// TIA Portal V19 export
FUNCTION_BLOCK "Arduino_Modbus"   // FB6, LAD
{ S7_Optimized_Access := 'TRUE' }
// v0.0.1 has not been tested
// stored: MemoryReserve 100, SetENOAutomatically false
   VAR_INPUT
      Proces_Item : Bool;
      Place_Item_Conveyor : Bool;
      Place_Item_Storage : Bool;
      Scrap_Item : Bool;
      Speed_Transport : Int := 10;
      Speed_Grinding : Int := 10;
      Grinding_Coordinates : Bool;
      Letter : DB_ANY;
   END_VAR
   VAR_OUTPUT
      Working : Bool;
      Done : Bool;
      Error : Bool;
      Reached_Coordinates : Bool;
   END_VAR
   VAR
      DISCONNECT : Bool;
      Address : TCON_IP_v4;
      ReceiveData : Array[0..5] of Int;
      SendData : Array[0..5] of Int;
   END_VAR
   // Address.InterfaceId := 64;
   // Address.ID := 1;
   // Address.ConnectionType := 11;
   // Address.ActiveEstablished := TRUE;
   // Address.RemoteAddress.ADDR[1] := 192;
   // Address.RemoteAddress.ADDR[2] := 168;
   // Address.RemoteAddress.ADDR[3] := 1;
   // Address.RemoteAddress.ADDR[4] := 61;
   // Address.RemotePort := 502;
   // Address.LocalPort := 502;
BEGIN

REGION Network 1: MB_CLIENT
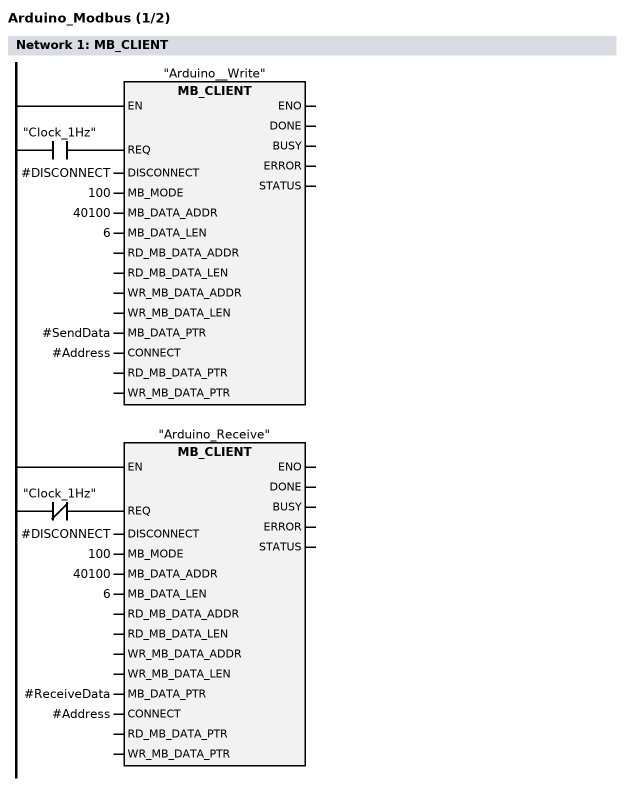
   RUNG wire#powerrail
      "Arduino__Write".MB_CLIENT(REQ := wire#w1, DISCONNECT := #DISCONNECT, MB_MODE := 100, MB_DATA_ADDR := 40100, MB_DATA_LEN := 6, RD_MB_DATA_ADDR :=, RD_MB_DATA_LEN :=, WR_MB_DATA_ADDR :=, WR_MB_DATA_LEN :=, MB_DATA_PTR := #SendData, CONNECT := #Address, RD_MB_DATA_PTR :=, WR_MB_DATA_PTR :=, DONE =>, BUSY =>, ERROR =>, STATUS =>)
   END_RUNG
   RUNG wire#powerrail
      Contact( "Clock_1Hz" )
   END_RUNG wire#w1
   RUNG wire#powerrail
      "Arduino_Receive".MB_CLIENT(REQ := wire#w2, DISCONNECT := #DISCONNECT, MB_MODE := 100, MB_DATA_ADDR := 40100, MB_DATA_LEN := 6, RD_MB_DATA_ADDR :=, RD_MB_DATA_LEN :=, WR_MB_DATA_ADDR :=, WR_MB_DATA_LEN :=, MB_DATA_PTR := #ReceiveData, CONNECT := #Address, RD_MB_DATA_PTR :=, WR_MB_DATA_PTR :=, DONE =>, BUSY =>, ERROR =>, STATUS =>)
   END_RUNG
   RUNG wire#powerrail
      I_Contact( "Clock_1Hz" )
   END_RUNG wire#w2
   // the same network as SCL:
   "Arduino__Write"(REQ := "Clock_1Hz",   // MB_CLIENT
                    DISCONNECT := #DISCONNECT,
                    MB_MODE := 100,
                    MB_DATA_ADDR := 40100,
                    MB_DATA_LEN := 6,
                    MB_DATA_PTR := #SendData,
                    CONNECT := #Address);
   "Arduino_Receive"(REQ := NOT "Clock_1Hz",   // MB_CLIENT
                     DISCONNECT := #DISCONNECT,
                     MB_MODE := 100,
                     MB_DATA_ADDR := 40100,
                     MB_DATA_LEN := 6,
                     MB_DATA_PTR := #ReceiveData,
                     CONNECT := #Address);
END_REGION

REGION Network 2: Send Data
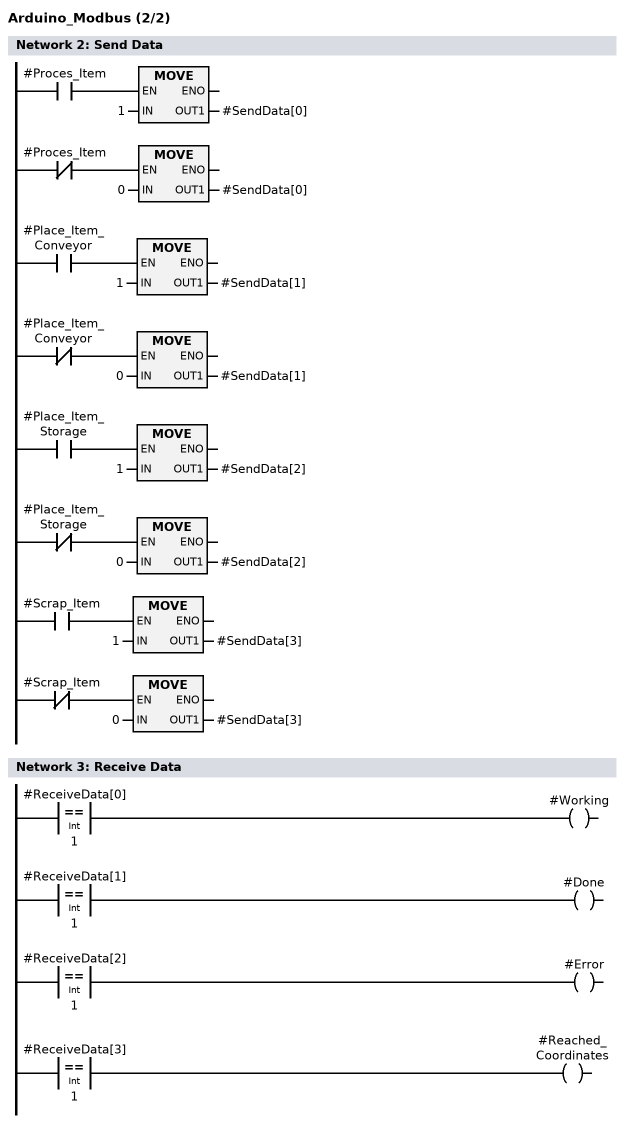
   RUNG wire#powerrail
      Contact( #Proces_Item )
      Move(in := 1, out1 => #SendData[0])
   END_RUNG
   RUNG wire#powerrail
      I_Contact( #Proces_Item )
      Move(in := 0, out1 => #SendData[0])
   END_RUNG
   RUNG wire#powerrail
      Contact( #Place_Item_Conveyor )
      Move(in := 1, out1 => #SendData[1])
   END_RUNG
   RUNG wire#powerrail
      I_Contact( #Place_Item_Conveyor )
      Move(in := 0, out1 => #SendData[1])
   END_RUNG
   RUNG wire#powerrail
      Contact( #Place_Item_Storage )
      Move(in := 1, out1 => #SendData[2])
   END_RUNG
   RUNG wire#powerrail
      I_Contact( #Place_Item_Storage )
      Move(in := 0, out1 => #SendData[2])
   END_RUNG
   RUNG wire#powerrail
      Contact( #Scrap_Item )
      Move(in := 1, out1 => #SendData[3])
   END_RUNG
   RUNG wire#powerrail
      I_Contact( #Scrap_Item )
      Move(in := 0, out1 => #SendData[3])
   END_RUNG
   // the same network as SCL:
   IF #Proces_Item THEN #SendData[0] := 1; END_IF;
   IF NOT #Proces_Item THEN #SendData[0] := 0; END_IF;
   IF #Place_Item_Conveyor THEN #SendData[1] := 1; END_IF;
   IF NOT #Place_Item_Conveyor THEN #SendData[1] := 0; END_IF;
   IF #Place_Item_Storage THEN #SendData[2] := 1; END_IF;
   IF NOT #Place_Item_Storage THEN #SendData[2] := 0; END_IF;
   IF #Scrap_Item THEN #SendData[3] := 1; END_IF;
   IF NOT #Scrap_Item THEN #SendData[3] := 0; END_IF;
END_REGION

REGION Network 3: Receive Data
   RUNG wire#powerrail
      { S7_Templates := "SrcType := Int" } EQ_Contact(in1 := #ReceiveData[0], in2 := 1)
      Coil( #Working )
   END_RUNG
   RUNG wire#powerrail
      { S7_Templates := "SrcType := Int" } EQ_Contact(in1 := #ReceiveData[1], in2 := 1)
      Coil( #Done )
   END_RUNG
   RUNG wire#powerrail
      { S7_Templates := "SrcType := Int" } EQ_Contact(in1 := #ReceiveData[2], in2 := 1)
      Coil( #Error )
   END_RUNG
   RUNG wire#powerrail
      { S7_Templates := "SrcType := Int" } EQ_Contact(in1 := #ReceiveData[3], in2 := 1)
      Coil( #Reached_Coordinates )
   END_RUNG
   // the same network as SCL:
   #Working := #ReceiveData[0] = 1;
   #Done := #ReceiveData[1] = 1;
   #Error := #ReceiveData[2] = 1;
   #Reached_Coordinates := #ReceiveData[3] = 1;
END_REGION
END_FUNCTION_BLOCK
